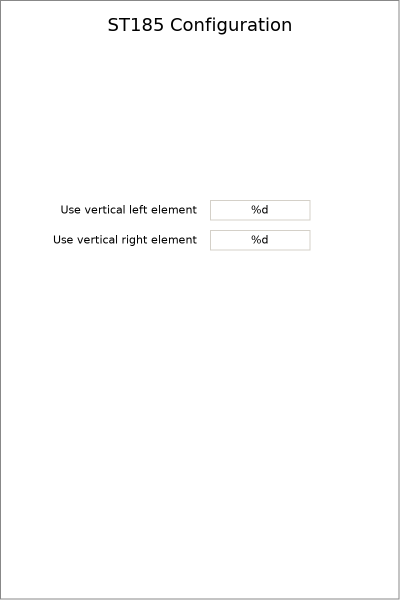
VISUALIZATION VISU_Recipe_ST185  // 400x600
    Label (0,5 400x40), "ST185 Configuration"
    Label (0,200 200x20), "Use vertical left element"
    Label (0,230 200x20), "Use vertical right element"
    Textfield (210,200 100x20), "%d", text variable: _20_AUTO.recipe.st185.xUseVerLeft
        OnMouseDown: write the text variable via Default
    Textfield (210,230 100x20), "%d", text variable: _20_AUTO.recipe.st185.xUseVerRight
        OnMouseDown: write the text variable via Default
END_VISUALIZATION

(* stored: Version 1.1.0.1, ProductVersion 3.1.4024.6
   Visu VISU_Recipe_ST185: Id {1aa6570a-0bb9-4327-b44f-684af424bdca} *)
